# EPICS substitutions: ek9000App/Db/EL4012.substitutions
file EL4012.template
{       pattern
        {
                TERMINAL,

        }
        {
        }
}
